# EPICS substitutions: utcaApp/Db/pbpm_pos_calc.substitutions
file db/scan_task.template {
    {}
}

file db/pbpm_pos_calc.template {
    {}
}

file db/pos_calc_adc.template {
    pattern {ADC, ADDR}
    {"A", 0}
    {"B", 1}
    {"C", 2}
    {"D", 3}
}

file db/pos_calc_rate.template {
    pattern {RATE, ADDR}
    {"TbT", 0}
    {"FAcq", 1}
    {"Monit", 2}
}
